{attribute 'qualified_only'}
{attribute 'strict'}
{attribute 'to_string'}
TYPE DUT_CircleMode :
(
	Border := 0,
	Center := 1,
	Radius := 2
);
END_TYPE

(* stored: Version 1.1.0.1
   EnumerationTextList DUT_CircleMode: Id {e3b49647-d147-4d35-a372-7d89a30539e3} *)
